TYPE UDT_BinBelt :
STRUCT
	bin: ARRAY [1..64] OF UDT_Bin;
END_STRUCT
END_TYPE

(* stored: Version 1.1.0.1, ProductVersion 3.1.4022.16
   DUT UDT_BinBelt: Id {f8cfd36c-cb99-4d44-9ad8-7cc516ce7441} *)
